// TIA Portal V19 export
DATA_BLOCK "FLUSHING VAVLE DB"   // DB63
{ S7_Optimized_Access := 'TRUE' }
// stored: MemoryReserve 100
   VAR
      "ABV 301" : Bool;
      "ABV 302" : Bool;
      "AGLV-301" : Bool;
      "AGLV-302" : Bool;
      "AGLV-401" : Bool;
      "AGLV-402" : Bool;
      "ABFV 501" : Bool;
      "ABFV 502" : Bool;
      "ABV 301 CLOSE VALVE" : Bool;
      "ABV 302 CLOSE VALVE" : Bool;
      "AGLV 301 CLOSE VALVE" : Bool;
      "AGLV 302 CLOSE VALVE" : Bool;
      "AGLV 401 CLOSE VALVE" : Bool;
      "AGLV-402 CLOSE VALVE" : Bool;
      "ABFV 501 CLOSE VALVE" : Bool;
      "ABFV 502 CLOSE VALVE" : Bool;
   END_VAR
BEGIN
END_DATA_BLOCK
